// TIA Portal V19 export
FUNCTION "Utgangssignaler" : Void   // FC1, LAD
{ S7_Optimized_Access := 'TRUE' }
// stored: SetENOAutomatically false
BEGIN

REGION Network 1
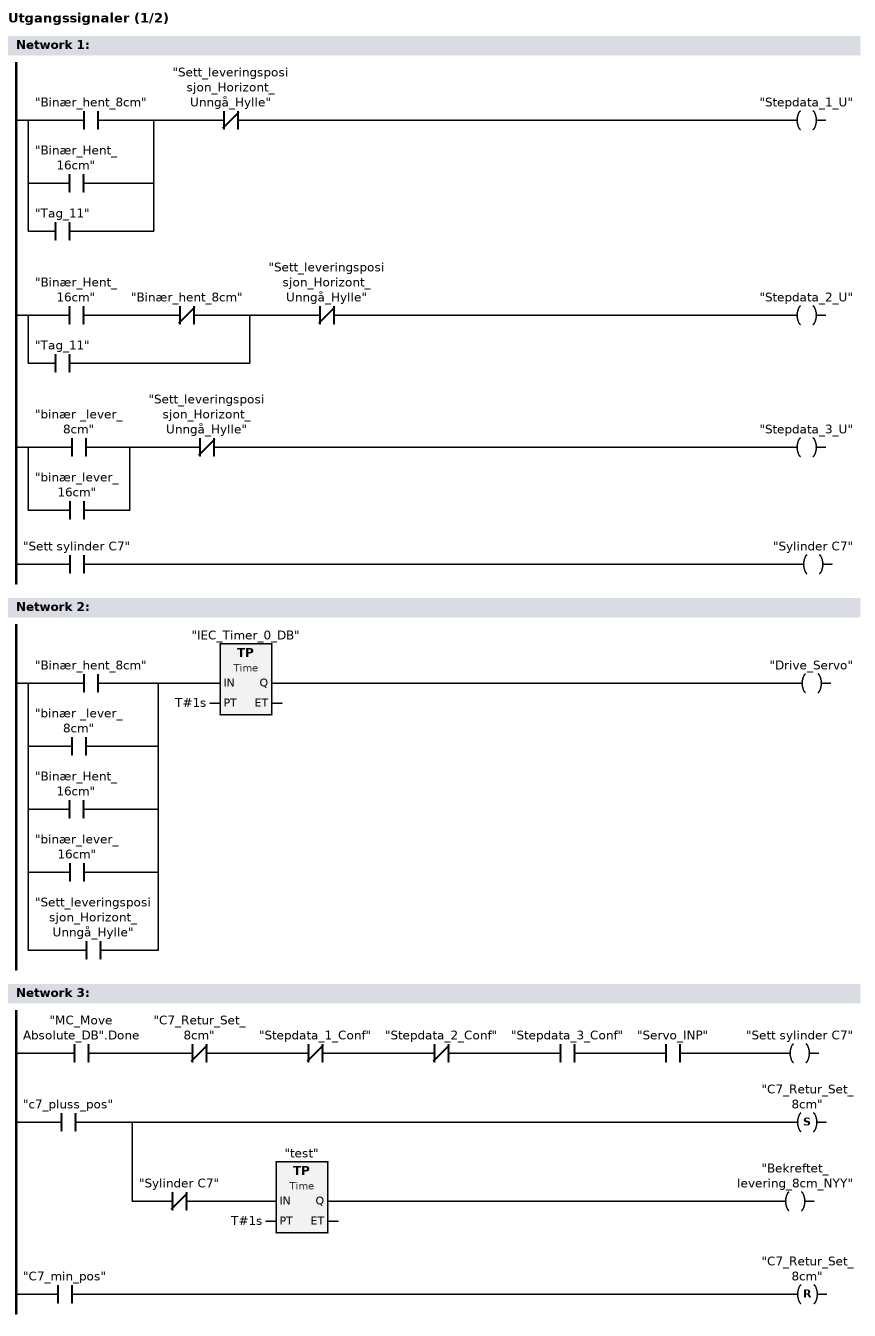
   RUNG wire#powerrail
      Contact( "Binær_hent_8cm" )
      wire#w1
      I_Contact( "Sett_leveringsposisjon_Horizont_Unngå_Hylle" )
      Coil( "Stepdata_1_U" )
   END_RUNG
   RUNG wire#powerrail
      Contact( "Binær_Hent_16cm" )
   END_RUNG wire#w1
   RUNG wire#powerrail
      Contact( "Tag_11" )
   END_RUNG wire#w1
   RUNG wire#powerrail
      Contact( "Binær_Hent_16cm" )
      I_Contact( "Binær_hent_8cm" )
      wire#w2
      I_Contact( "Sett_leveringsposisjon_Horizont_Unngå_Hylle" )
      Coil( "Stepdata_2_U" )
   END_RUNG
   RUNG wire#powerrail
      Contact( "Tag_11" )
   END_RUNG wire#w2
   RUNG wire#powerrail
      Contact( "binær _lever_8cm" )
      wire#w3
      I_Contact( "Sett_leveringsposisjon_Horizont_Unngå_Hylle" )
      Coil( "Stepdata_3_U" )
   END_RUNG
   RUNG wire#powerrail
      Contact( "binær_lever_16cm" )
   END_RUNG wire#w3
   RUNG wire#powerrail
      Contact( "Sett sylinder C7" )
      Coil( "Sylinder C7" )
   END_RUNG
   // the same network as SCL:
   "Stepdata_1_U" := ("Binær_hent_8cm" OR "Binær_Hent_16cm" OR "Tag_11") AND NOT "Sett_leveringsposisjon_Horizont_Unngå_Hylle";
   "Stepdata_2_U" := (("Binær_Hent_16cm" AND NOT "Binær_hent_8cm") OR "Tag_11") AND NOT "Sett_leveringsposisjon_Horizont_Unngå_Hylle";
   "Stepdata_3_U" := ("binær _lever_8cm" OR "binær_lever_16cm") AND NOT "Sett_leveringsposisjon_Horizont_Unngå_Hylle";
   "Sylinder C7" := "Sett sylinder C7";
END_REGION

REGION Network 2
   RUNG wire#powerrail
      Contact( "Binær_hent_8cm" )
      wire#w1
      { S7_Templates := "time_type := Time" } "IEC_Timer_0_DB".TP(pt := T#1s, et =>)
      Coil( "Drive_Servo" )
   END_RUNG
   RUNG wire#powerrail
      Contact( "binær _lever_8cm" )
   END_RUNG wire#w1
   RUNG wire#powerrail
      Contact( "Binær_Hent_16cm" )
   END_RUNG wire#w1
   RUNG wire#powerrail
      Contact( "binær_lever_16cm" )
   END_RUNG wire#w1
   RUNG wire#powerrail
      Contact( "Sett_leveringsposisjon_Horizont_Unngå_Hylle" )
   END_RUNG wire#w1
   // the same network as SCL:
   "IEC_Timer_0_DB".TP(IN := "Binær_hent_8cm" OR "binær _lever_8cm" OR "Binær_Hent_16cm" OR "binær_lever_16cm" OR "Sett_leveringsposisjon_Horizont_Unngå_Hylle",
                       PT := T#1s);
   "Drive_Servo" := "IEC_Timer_0_DB".Q;
END_REGION

REGION Network 3
   RUNG wire#powerrail
      Contact( "MC_MoveAbsolute_DB".Done )
      I_Contact( "C7_Retur_Set_8cm" )
      I_Contact( "Stepdata_1_Conf" )
      I_Contact( "Stepdata_2_Conf" )
      Contact( "Stepdata_3_Conf" )
      Contact( "Servo_INP" )
      Coil( "Sett sylinder C7" )
   END_RUNG
   RUNG wire#powerrail
      Contact( "c7_pluss_pos" )
      wire#w1
      S_Coil( "C7_Retur_Set_8cm" )
   END_RUNG
   RUNG wire#w1
      I_Contact( "Sylinder C7" )
      { S7_Templates := "time_type := Time" } "test".TP(pt := T#1s, et =>)
      Coil( "Bekreftet_levering_8cm_NYY" )
   END_RUNG
   RUNG wire#powerrail
      Contact( "C7_min_pos" )
      R_Coil( "C7_Retur_Set_8cm" )
   END_RUNG
   // the same network as SCL:
   "Sett sylinder C7" := "MC_MoveAbsolute_DB".Done AND NOT "C7_Retur_Set_8cm" AND NOT "Stepdata_1_Conf" AND NOT "Stepdata_2_Conf" AND "Stepdata_3_Conf" AND "Servo_INP";
   IF "c7_pluss_pos" THEN "C7_Retur_Set_8cm" := TRUE; END_IF;
   "test".TP(IN := "c7_pluss_pos" AND NOT "Sylinder C7", PT := T#1s);
   "Bekreftet_levering_8cm_NYY" := "test".Q;
   IF "C7_min_pos" THEN "C7_Retur_Set_8cm" := FALSE; END_IF;
END_REGION

REGION Network 4
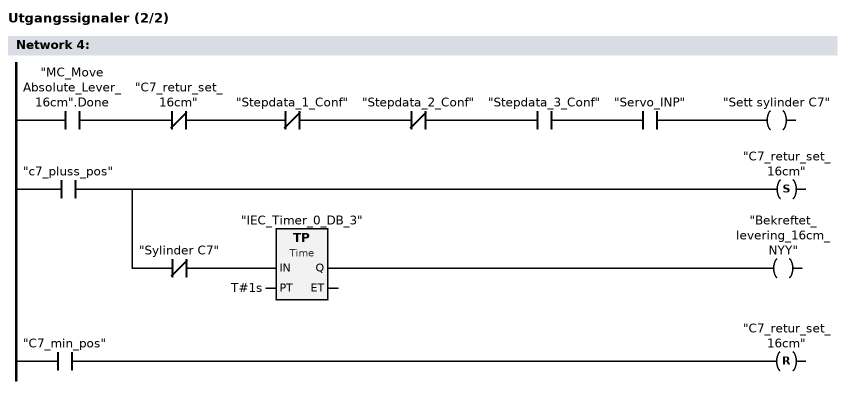
   RUNG wire#powerrail
      Contact( "MC_MoveAbsolute_Lever_16cm".Done )
      I_Contact( "C7_retur_set_16cm" )
      I_Contact( "Stepdata_1_Conf" )
      I_Contact( "Stepdata_2_Conf" )
      Contact( "Stepdata_3_Conf" )
      Contact( "Servo_INP" )
      Coil( "Sett sylinder C7" )
   END_RUNG
   RUNG wire#powerrail
      Contact( "c7_pluss_pos" )
      wire#w1
      S_Coil( "C7_retur_set_16cm" )
   END_RUNG
   RUNG wire#w1
      I_Contact( "Sylinder C7" )
      { S7_Templates := "time_type := Time" } "IEC_Timer_0_DB_3".TP(pt := T#1s, et =>)
      Coil( "Bekreftet_levering_16cm_NYY" )
   END_RUNG
   RUNG wire#powerrail
      Contact( "C7_min_pos" )
      R_Coil( "C7_retur_set_16cm" )
   END_RUNG
   // the same network as SCL:
   "Sett sylinder C7" := "MC_MoveAbsolute_Lever_16cm".Done AND NOT "C7_retur_set_16cm" AND NOT "Stepdata_1_Conf" AND NOT "Stepdata_2_Conf" AND "Stepdata_3_Conf" AND "Servo_INP";
   IF "c7_pluss_pos" THEN "C7_retur_set_16cm" := TRUE; END_IF;
   "IEC_Timer_0_DB_3".TP(IN := "c7_pluss_pos" AND NOT "Sylinder C7", PT := T#1s);
   "Bekreftet_levering_16cm_NYY" := "IEC_Timer_0_DB_3".Q;
   IF "C7_min_pos" THEN "C7_retur_set_16cm" := FALSE; END_IF;
END_REGION
END_FUNCTION
